{attribute 'qualified_only'}
VAR_GLOBAL
	
	Mode: Modes;
END_VAR

(* stored: Version 1.1.0.1, ProductVersion 3.1.4024.9
   GVL GVL: Id {46d428ad-1ef1-4941-a8be-12cc2c082151} *)
